# EPICS autosave request: support/dxp-s55/dxpApp/Db/dxpHighLevel_settings.req
$(P)$(R)PeakingTime
$(P)$(R)TriggerThreshold
$(P)$(R)BaselineThreshold
$(P)$(R)BaselineCutPercent
$(P)$(R)BaselineCutEnable
$(P)$(R)BaselineFilterLength
$(P)$(R)EnergyThreshold
$(P)$(R)ADCPercentRule
$(P)$(R)MaxEnergy
$(P)$(R)PreampGain
$(P)$(R)DetectorPolarity
$(P)$(R)ResetDelay
$(P)$(R)GapTime
$(P)$(R)TriggerPeakingTime
$(P)$(R)TriggerGapTime
$(P)$(R)MaxWidth
$(P)$(R)PresetMode
$(P)$(R)PresetEvents
$(P)$(R)PresetTriggers
$(P)$(R)TraceMode
$(P)$(R)TraceTime
$(P)$(R)NumSCAs
